Staubli VAL3: getByteAt.pgx

public program getByteAt(num x_nByteIndex, num& x_nBuffer[], num& x_nRes)
begin

  x_nRes=x_nBuffer[x_nByteIndex]

end
